Staubli VAL3: call.pjx

Parameters version=s7.1 stackSize=5000 millimeterUnit=true
Program file=start.pgx
Program file=stop.pgx
Data file=call.dtx
